INTERFACE Test_interface

METHOD MoveAllToPosition : Test_interface
VAR_INPUT

	DestinationPosition		: LREAL;		// position on track for all shuttles to move towards	

END_VAR
END_METHOD

END_INTERFACE

(* stored: Version 1.1.0.1, ProductVersion 3.1.4024.9
   Itf Test_interface: Id {9cc4a2ad-2506-4bdd-acf3-bfbfde25ab77}
   Method MoveAllToPosition: Id {745a52d9-fa71-49ff-868a-52a3293e2e2d} *)
